Staubli VAL3: StaubliUI.pjx

--- StaubliUI.pjx ---
Parameters version=s7.3 stackSize=15000 millimeterUnit=true
Program file=Bool_Edit.pgx
Program file=BoolMess_Edit.pgx
Program file=Control_Action.pgx
Program file=Control_AxisPar.pgx
Program file=Control_BatPara.pgx
Program file=Control_BatPrt.pgx
Program file=Control_BatSpd.pgx
Program file=Control_Bottom.pgx
Program file=Control_BottomS.pgx
Program file=Control_CPreset.pgx
Program file=Control_Joint.pgx
Program file=Control_Lable.pgx
Program file=Control_Left.pgx
Program file=Control_LeftCut.pgx
Program file=Control_LeftS.pgx
Program file=Control_List.pgx
Program file=Control_List1S.pgx
Program file=Control_ListBS.pgx
Program file=Control_ListCls.pgx
Program file=Control_ListMC.pgx
Program file=Control_ListMCD.pgx
Program file=Control_ListS.pgx
Program file=Control_Loffset.pgx
Program file=Control_MCShow.pgx
Program file=Control_Mess.pgx
Program file=Control_Panel.pgx
Program file=Control_PanelB.pgx
Program file=Control_PanelD.pgx
Program file=Control_PanelMd.pgx
Program file=Control_PanelS.pgx
Program file=Control_PanelXY.pgx
Program file=Control_PanTitl.pgx
Program file=Control_Para.pgx
Program file=Control_Para1.pgx
Program file=Control_PatMove.pgx
Program file=Control_Point.pgx
Program file=Control_Preset.pgx
Program file=Control_Recipe.pgx
Program file=Control_Remote.pgx
Program file=Control_Scara.pgx
Program file=Control_Timer.pgx
Program file=Control_Traj.pgx
Program file=Control_YesNO.pgx
Program file=Float_Edit.pgx
Program file=Form_4jHome.pgx
Program file=Form_6jHome.pgx
Program file=Form_Action.pgx
Program file=Form_Bye.pgx
Program file=Form_Config.pgx
Program file=Form_LabelList.pgx
Program file=Form_Main.pgx
Program file=Form_MainS.pgx
Program file=Form_Panel.pgx
Program file=Form_Panel4P.pgx
Program file=Form_PanelBool.pgx
Program file=Form_PanelJoint.pgx
Program file=Form_PanelList.pgx
Program file=Form_PanelPoint.pgx
Program file=Form_PanelStr.pgx
Program file=Form_Patten.pgx
Program file=Form_PattenD.pgx
Program file=Form_PattenS.pgx
Program file=Form_Prod.pgx
Program file=Form_Product.pgx
Program file=Form_ScaraRobot.pgx
Program file=Form_SelSharp.pgx
Program file=Form_Simulation.pgx
Program file=Form_Welcome.pgx
Program file=Int_Edit.pgx
Program file=Int_EditS.pgx
Program file=Key_ListBase.pgx
Program file=Key_ListMC.pgx
Program file=ReadMe.pgx
Program file=Sel_Edit.pgx
Program file=start.pgx
Program file=stop.pgx
Program file=Str_Edit.pgx
Program file=Str_SplitChar.pgx
Program file=Str_SplitComma.pgx
Data file=StaubliUI.dtx

--- StaubliUI.dtx ---
mdesc mNomSpeed
num nPanelLTopX
num nPanelLTopY
num nPanelWidthX
num nPanelLengthY
string sBuff
string sData

--- Control_AxisPar.pgx ---
public program Control_AxisPar(num& x_nPos, num& x_nSpeed, num& x_nPrecent, num& x_nJogSpeed, bool x_bTraj)
  local string l_sItem[6]
  local num l_nNum
  local num l_nKey
  local num l_nData[6]
  local num l_nSelectIndex
begin
  //为lasman3.0进行配置
  //修改点位的参数


  //通过局部变量来实现内部存储


  l_nData[0]=x_nPos
  l_nData[1]=x_nSpeed
  l_nData[2]=x_nPrecent
  l_nData[3]=x_nJogSpeed

  l_sItem[0]="位置mm   :"+toString(".3",l_nData[0])
  l_sItem[1]="速度m/min:"+toString(".3",l_nData[1])
  l_sItem[2]="比例分度 :"+toString(".3",l_nData[2])
  l_sItem[3]="点动速度 :"+toString(".3",l_nData[3])
  call Control_BottomS(",,,,,,取消,确定")

  call Control_PanelXY(8,0,17,4)
  call Control_Panel("参数")
  call Control_List(l_sItem,l_nSelectIndex)


  //按键响应
  while true
    l_nKey=getKey()

    switch l_nKey
      case 261
        l_nSelectIndex=max(0,l_nSelectIndex-1)
      break

      case 266
        if x_bTraj
          l_nSelectIndex=min(1,l_nSelectIndex+1)
        else
           l_nSelectIndex=min(3,l_nSelectIndex+1)
        endIf

      break

      case 278

        x_nPos=l_nData[0]
        x_nSpeed=l_nData[1]
        x_nPrecent=l_nData[2]
        x_nJogSpeed=l_nData[3]
        cls()
        return
      break


      case 277,255
        cls()
        return
      break



      case 270

        call Float_Edit(l_nData[l_nSelectIndex],nPanelLTopX+11,l_nSelectIndex+nPanelLTopY+1)


        l_nData[l_nSelectIndex]=max(0,l_nData[l_nSelectIndex])
        l_nData[3]=min(100,max(0,l_nData[3]))
      break

    endSwitch

    if l_nKey!=-1
      l_sItem[0]="位置mm   :"+toString(".3",l_nData[0])
      l_sItem[1]="速度m/min:"+toString(".3",l_nData[1])
      l_sItem[2]="比例分度 :"+toString(".3",l_nData[2])
      l_sItem[3]="点动速度 :"+toString(".3",l_nData[3])
      call Control_List(l_sItem,l_nSelectIndex)

    endIf






  endWhile

end

--- Control_BatSpd.pgx ---
public program Control_BatSpd(num& x_nFrom, num& x_nTo, num& x_nSpeed, num& x_nAcc)
  local string l_sItem[4]
  local num l_nNum
  local num l_nKey
  local num l_nData[6]
  local num l_nSelectIndex
begin

  //为lasman3.0进行配置
  //批处理速度


  l_nData[0]=x_nFrom
  l_nData[1]=x_nTo
  l_nData[2]=100
  l_nData[3]=15
  l_sItem[0]="开始序号:"+toString("",l_nData[0])
  l_sItem[1]="结束序号:"+toString("",l_nData[1])
  l_sItem[2]="速度    :"+toString("",l_nData[2])
  l_sItem[3]="加速度  :"+toString("",l_nData[3])



  call Control_BottomS(",,,,,,取消,确定")
  call Control_PanelXY(8,0,15,4)
  call Control_Panel("批处理速度")
  call Control_List(l_sItem,l_nSelectIndex)
  while true
    l_nKey=getKey()

    switch l_nKey
      case 261
        l_nSelectIndex=max(0,l_nSelectIndex-1)
      break

      case 266
        l_nSelectIndex=min(l_nSelectIndex+1,3)
      break

      case 278
        x_nFrom=l_nData[0]
        x_nTo=l_nData[1]
        x_nSpeed=l_nData[2]
        x_nAcc=l_nData[3]
        cls()
        return
      break


      case 277,255

        cls()
        return
      break

      case 270

        call Float_Edit(l_nData[l_nSelectIndex],nPanelLTopX+7,l_nSelectIndex+nPanelLTopY+1)
      break

    endSwitch

    if l_nKey!=-1
  l_sItem[0]="开始序号:"+toString("",l_nData[0])
  l_sItem[1]="结束序号:"+toString("",l_nData[1])
  l_sItem[2]="速度    :"+toString("",l_nData[2])
  l_sItem[3]="加速度  :"+toString("",l_nData[3])
      call Control_List(l_sItem,l_nSelectIndex)

    endIf






  endWhile





end

--- Control_CPreset.pgx ---
public program Control_CPreset(num& x_nPreset[] (dimensions=2), trsf& x_trCut[], num x_nMax, num x_nIndex)
  local string l_sItem[6]
  local num l_nNum
  local num l_nKey
  local num l_nData[5]
  local num l_nIndex
  local num l_nBuff
  local bool l_bFirst
begin

  //为lasman3.0进行定制
  //修改工艺参数


  //  //把传入参数临时存储
  //  l_nIndex=x_trCut[x_nIndex].x
  //  for l_nNum=0 to 4
  //    l_nData[l_nNum]=x_nPreset[l_nIndex,l_nNum]
  //  endFor
  //
  //  //界面初始化
  //      l_sItem[0]="工艺号  :"+toString("",l_nIndex)
  //      l_sItem[1]="激光功率  :"+toString("",l_nData[0])
  //      l_sItem[2]="气体压力  :"+toString("",l_nData[1])
  //      l_sItem[3]="占空比频率:"+toString("",l_nData[2])
  //      l_sItem[4]="激光占空比:"+toString("",l_nData[3])
  //      l_sItem[5]="随动高度  :"+toString("",l_nData[4])
  //      call Control_List(l_sItem,l_nBuff)
   l_nIndex=x_trCut[x_nIndex].x
  call Control_BottomS(",,,,,,退出,应用")
  call Control_PanelXY(8,0,15,6)
  call Control_Panel(toString("",x_nIndex)+":工艺值")
  call Control_List(l_sItem,l_nBuff)
  //按键响应
  while true
    l_nKey=getKey()

    switch l_nKey
      case 261
        l_nIndex=max(1,l_nIndex-1)
        //l_nSelectIndex=max(0,l_nSelectIndex-1)
      break

      case 266
        l_nIndex=min(50,l_nIndex+1)
        // l_nSelectIndex=min(l_nSelectIndex+1,5)
      break

      case 264
        x_nIndex=max(0,x_nIndex-1)


      break



      case 268
        x_nIndex=min(x_nMax-1,x_nIndex+1)
         l_nIndex=x_trCut[x_nIndex].x
      break





      case 278
        //        for l_nNum=0 to 4
        //          x_nPreset[x_nIndex,l_nNum]=min(max(l_nData[l_nNum],0),100)
        //      x.x=l_nIndex
        x_trCut[x_nIndex].x=l_nIndex
     //   return
      l_nIndex=x_trCut[x_nIndex].x
      break


      case 277
        return
      break

      //      case 270
      //        call Float_Edit(l_nData[l_nSelectIndex],nPanelLTopX+12,l_nSelectIndex+nPanelLTopY+1)
      //        l_nData[l_nSelectIndex]=min(max(l_nData[l_nSelectIndex],0),100)
      //      break

    endSwitch

    if l_nKey!=-1 or !l_bFirst
      l_bFirst=true

      for l_nNum=0 to 4
        l_nData[l_nNum]=x_nPreset[l_nIndex,l_nNum]
      endFor
      for l_nNum=0 to 4
        l_nData[l_nNum]=x_nPreset[l_nIndex,l_nNum]
      endFor
         call Control_PanTitl(toString("",x_nIndex+1)+"点:工艺值")
      l_sItem[0]="工艺号    :"+toString("",l_nIndex)
      l_sItem[1]="激光功率  :"+toString("",l_nData[0])
      l_sItem[2]="气体压力  :"+toString("",l_nData[1])
      l_sItem[3]="占空比频率:"+toString("",l_nData[2])
      l_sItem[4]="激光占空比:"+toString("",l_nData[3])
      l_sItem[5]="随动高度  :"+toString("",l_nData[4])
      call Control_List(l_sItem,l_nBuff)

    endIf







  endWhile





end

--- Control_ListCls.pgx ---
program Control_ListCls()
  local num l_nIndex
begin

  //说明：
  //函数功能：把方框中进行清空




  //对方框的定义进行赋初值
  if nPanelLengthY<=0 and nPanelLTopX<=0 and nPanelLTopY<=0 and nPanelWidthX<=0
    call Control_PanelXY(20,0,18,11)
  endIf

  //清空列表
  setTextMode(0)
  for l_nIndex=0 to nPanelLengthY-1
    gotoxy(nPanelLTopX+1,nPanelLTopY+l_nIndex+1)
    put(left("                                               ",nPanelWidthX))
  endFor

  //参数判断  对于选择项的判断
  // x_nSelectItem=min(max(0,x_nSelectItem),nPanelLengthY-1)


end

--- Control_ListMC.pgx ---
public program Control_ListMC(bool& x_bMC[], num& x_nSelectItem, num x_nText)
  local num l_nIndex
  local bool l_bRes
  local string l_sText
  local num l_nFrist
begin
  //说明：
  //函数功能：在划定的框内，把选中项给显示出来
  //l_nFirst  在列表中第一个显示的项的序号
  //x_nSelectItem  被选中的项的序号
  //l_nCount 合法列表项的项总数，如何数组中间为空，则可能被截断

  l_nFrist=0
  x_nSelectItem=min(max(0,x_nSelectItem),size(x_bMC)-1)
  if x_nSelectItem>=nPanelLengthY
    l_nFrist=x_nSelectItem-nPanelLengthY+1
  endIf


  //把列表给画出来
  for l_nIndex=0 to min(nPanelLengthY-1,size(x_bMC)-l_nFrist)
    gotoxy(nPanelLTopX+1,nPanelLTopY+l_nIndex+1)
    //选中项变成黑色


    //MOVEL
    if !x_bMC[l_nIndex+l_nFrist]
      if l_nIndex+l_nFrist==x_nSelectItem

        setTextMode(1)
      else
        setTextMode(0)
      endIf
      put(left(toString("",l_nIndex+l_nFrist+1)+"       ",5 )+left("MOVEL             ",nPanelWidthX-5))
    else

      //MOVEC
      setTextMode(0)
      put(left("                                               ",nPanelWidthX))
      gotoxy(nPanelLTopX+1,nPanelLTopY+l_nIndex+1)
      if l_nIndex+l_nFrist!=x_nSelectItem
        put(left(toString("",l_nIndex+l_nFrist+1)+"       ",5 )+left("MOVEC Pc Pt              ",nPanelWidthX-5))
      else
        if x_nText==0
          setTextMode(1)
        else
          setTextMode(0)
        endIf
        put(left(toString("",l_nIndex+l_nFrist+1)+"       ",5 )+"MOVEC")
        gotoxy(nPanelLTopX+12,nPanelLTopY+l_nIndex+1)
        if x_nText==1

          setTextMode(1)
        else
          setTextMode(0)
        endIf
        put("Pc")
        //目标点
        gotoxy(nPanelLTopX+15,nPanelLTopY+l_nIndex+1)

        if x_nText==2
          setTextMode(1)
        else
          setTextMode(0)
        endIf
        put("Pt")
      endIf
    endIf
  endFor

  setTextMode(0)
  while l_nIndex< nPanelLengthY
    gotoxy(nPanelLTopX+1,nPanelLTopY+l_nIndex+1)
    put(left("                          ",nPanelWidthX-2))
    l_nIndex=l_nIndex+1
  endWhile

end

--- Control_Loffset.pgx ---
public program Control_Loffset(num& x_nFrom, num& x_nTo)
  local string l_sItem[2]
  local num l_nNum
  local num l_nKey
  local num l_nData[6]
  local num l_nSelectIndex
begin

  //为lasman3.0配置
  //局部偏差
l_nData[0]=x_nFrom
l_nData[1]=x_nTo

  l_sItem[0]="开始    :"+toString("",l_nData[0])
  l_sItem[1]="停止    :"+toString("",l_nData[1])
  call Control_BottomS(",,,,,,取消,确定")
  call Control_PanelXY(8,0,15,6)
  call Control_Panel("局部偏差值")
  call Control_List(l_sItem,l_nSelectIndex)
  while true
    l_nKey=getKey()

    switch l_nKey
      case 261
        l_nSelectIndex=max(0,l_nSelectIndex-1)
      break

      case 266
        l_nSelectIndex=min(l_nSelectIndex+1,1)
      break

      case 278
          x_nFrom=l_nData[0]
          x_nTo=l_nData[1]
         cls()
        return
      break


      case 277,255

        cls()
        return
      break

      case 270
        call Float_Edit(l_nData[l_nSelectIndex],nPanelLTopX+7,l_nSelectIndex+nPanelLTopY+1)
      break

    endSwitch

    if l_nKey!=-1
  l_sItem[0]="开始    :"+toString("",l_nData[0])
  l_sItem[1]="停止    :"+toString("",l_nData[1])
      call Control_List(l_sItem,l_nSelectIndex)

    endIf






  endWhile





end

--- Control_MCShow.pgx ---
public program Control_MCShow(num x_nIndex, num x_nMoveType)
  local string l_sS[3]
begin

  //lasman3.0
  //为圆弧进行配置

  if x_nMoveType>2 or x_nMoveType<1
    return
  endIf
  l_sS[0]=toString("",x_nIndex+1)+"."+"MoveC "
  l_sS[1]=toString("",1)+" "
  l_sS[2]=left(" "+toString("",2)+"       ",nPanelWidthX-len(l_sS[0])-len(l_sS[1]))
  setTextMode(0)
  gotoxy(nPanelLTopX+1,min(nPanelLengthY,x_nIndex+1))
  put(l_sS[0])
  setTextMode(sel(x_nMoveType==1,1,0))
  put(l_sS[1])
  setTextMode(sel(x_nMoveType==1,0,1))
  put(l_sS[2])


  setTextMode(0)

end

--- Control_PanelB.pgx ---
public program Control_PanelB(string x_sLeftTitle, string x_sRightTitle)
begin

  //画左右两个方框

  call Control_PanelS(x_sLeftTitle,0,0,18,11)

  call Control_PanelS(x_sRightTitle,20,0,18,11)

end

--- Control_PanelS.pgx ---
public program Control_PanelS(string x_sTitle, num x_nLTopX, num x_nLTopY, num x_nWidthX, num x_nLengthY)
  local num l_nIndex
begin
  //画有标题的框



  //设定框的位置与大小
  call Control_PanelXY(x_nLTopX,x_nLTopY,x_nWidthX,x_nLengthY)

  //文本显示状况进行设定
   call Control_Panel(x_sTitle)



end

--- Control_Para1.pgx ---
public program Control_Para1(trsf& x_trTrsf, bool& x_bRes, bool x_bCut, num x_nType)
  local string l_sItem[6]
  local num l_nNum
  local num l_nKey
  local num l_nData[6]
  local num l_nSelectIndex
begin
  //为lasman3.0进行配置
  //修改点位的参数


  //通过局部变量来实现内部存储
  l_nData[3]=x_trTrsf.x
  l_nData[4]=x_trTrsf.y
  l_nData[0]=x_trTrsf.z
  l_nData[1]=x_trTrsf.rx

  l_nData[2]=x_trTrsf.ry
  l_nData[5]=x_trTrsf.rz
  l_nNum=sel(x_bRes,1,0)

  //界面初始化
  resize(sData,1,2)
  if x_bCut

    sData[0]="直线"
    sData[1]="圆弧"
    l_sItem[0]="速度(mm/s:"+toString(".3",l_nData[0])
    l_sItem[1]="加速度(%):"+toString(".3",l_nData[1])
    l_sItem[2]="BLend(mm):"+toString(".3",l_nData[2])
    l_sItem[3]="工艺     :"+toString(".3",l_nData[3])
    l_sItem[4]="动作     :"+toString(".3",l_nData[4])
    l_sItem[5]="圆弧/直线:"+sData[l_nNum]

  else
    sData[0]="MoveJ"
    sData[1]="MoveL"
    l_sItem[0]="速度(mm/s:"+toString(".3",l_nData[0])
    l_sItem[1]="加速度(%):"+toString(".3",l_nData[1])
    l_sItem[2]="关节/直线:"+sData[l_nNum]

  endIf

  call Control_BottomS(",,,,,,取消,确定")
  if x_bCut
    if x_nType!=10
      call Control_PanelXY(8,0,18,5)
    else
      call Control_PanelXY(8,0,18,6)
    endIf
  else
    call Control_PanelXY(8,0,17,3)
  endIf
  call Control_Panel("参数")
  call Control_List(l_sItem,l_nSelectIndex)


  //按键响应
  while true
    l_nKey=getKey()

    switch l_nKey
      case 261
        l_nSelectIndex=max(0,l_nSelectIndex-1)
      break

      case 266
        if x_bCut
          if x_nType==10
            l_nSelectIndex=min(l_nSelectIndex+1,5)
          else
            l_nSelectIndex=min(l_nSelectIndex+1,4)
          endIf
        else
          l_nSelectIndex=min(l_nSelectIndex+1,2)
        endIf
      break

      case 278
        x_trTrsf.x=l_nData[3]
        x_trTrsf.y=l_nData[4]
        x_trTrsf.z=l_nData[0]
        x_trTrsf.rx=l_nData[1]

        x_trTrsf.ry=l_nData[2]
        x_trTrsf.rz=l_nData[5]
        x_bRes=(l_nNum==1)
        cls()
        return
      break


      case 277,255
        cls()
        return
      break



      case 270
        if (l_nSelectIndex==2 and !x_bCut) or (l_nSelectIndex==5 and x_bCut)
          call Sel_Edit(l_nNum,nPanelLTopX+11,l_nSelectIndex+nPanelLTopY+1,sData)

        else
          call Float_Edit(l_nData[l_nSelectIndex],nPanelLTopX+11,l_nSelectIndex+nPanelLTopY+1)
        endIf
      break

    endSwitch

    if l_nKey!=-1
      if x_bCut

        sData[0]="直线"
        sData[1]="圆弧"
        l_sItem[0]="速度(mm/s:"+toString(".3",l_nData[0])
        l_sItem[1]="加速度(%):"+toString(".3",l_nData[1])
        l_sItem[2]="BLend(mm):"+toString(".3",l_nData[2])
        l_sItem[3]="工艺     :"+toString(".3",l_nData[3])
        l_sItem[4]="动作     :"+toString(".3",l_nData[4])
        l_sItem[5]="圆弧/直线:"+sData[l_nNum]

      else
        sData[0]="MoveJ"
        sData[1]="MoveL"
        l_sItem[0]="速度(mm/s:"+toString(".3",l_nData[0])
        l_sItem[1]="加速度(%):"+toString(".3",l_nData[1])
        l_sItem[2]="关节/直线:"+sData[l_nNum]

      endIf
      call Control_List(l_sItem,l_nSelectIndex)

    endIf






  endWhile

end

--- Control_Point.pgx ---
public program Control_Point(pointRx& x_pP)
  local string l_sItem[6]
  local num l_nNum
  local num l_nKey
  local num l_nData[6]
  local num l_nSelectIndex
begin

  //修改点位的 Point

  l_nData[0]=x_pP.trsf.x
  l_nData[1]=x_pP.trsf.y
  l_nData[2]=x_pP.trsf.z
  l_nData[3]=x_pP.trsf.rx
  l_nData[4]=x_pP.trsf.ry
  l_nData[5]=x_pP.trsf.rz

  l_sItem[0]="X    :"+toString(".3",l_nData[0])
  l_sItem[1]="y    :"+toString(".3",l_nData[1])
  l_sItem[2]="Z    :"+toString(".3",l_nData[2])
  l_sItem[3]="RX   :"+toString(".3",l_nData[3])
  l_sItem[4]="RY   :"+toString(".3",l_nData[4])
  l_sItem[5]="RZ   :"+toString(".3",l_nData[5])

  call Control_BottomS(",,,,,,取消,确定")
  call Control_PanelXY(8,0,15,6)
  call Control_Panel("Point值")
  call Control_List(l_sItem,l_nSelectIndex)
  while true
    l_nKey=getKey()

    switch l_nKey
      case 261
        l_nSelectIndex=max(0,l_nSelectIndex-1)
      break

      case 266
        l_nSelectIndex=min(l_nSelectIndex+1,5)
      break

      case 278
        x_pP.trsf.x=l_nData[0]
        x_pP.trsf.y=l_nData[1]
        x_pP.trsf.z=l_nData[2]
        x_pP.trsf.rx=l_nData[3]
        x_pP.trsf.ry=l_nData[4]
        x_pP.trsf.rz=l_nData[5]
        cls()
        return
      break


      case 277,255

        cls()
        return
      break

      case 270
        call Float_Edit(l_nData[l_nSelectIndex],nPanelLTopX+7,l_nSelectIndex+nPanelLTopY+1)
      break

    endSwitch

    if l_nKey!=-1
      l_sItem[0]="X    :"+toString(".3",l_nData[0])
      l_sItem[1]="y    :"+toString(".3",l_nData[1])
      l_sItem[2]="Z    :"+toString(".3",l_nData[2])
      l_sItem[3]="RX   :"+toString(".3",l_nData[3])
      l_sItem[4]="RY   :"+toString(".3",l_nData[4])
      l_sItem[5]="RZ   :"+toString(".3",l_nData[5])
      call Control_List(l_sItem,l_nSelectIndex)

    endIf






  endWhile





end

--- Control_Remote.pgx ---
public program Control_Remote(num& x_nMode, num& x_nCycleCount)
  local string l_sItem[2]
  local num l_nNum
  local num l_nKey
  local num l_nData[2]
  local num l_nSelectIndex
  local string l_sSMess[6]
begin

  //为lasman3.0进行配置
  //主要是远程选择界面



  l_nData[0]=max(round(x_nMode),0)
  l_nData[1]=max(round(x_nCycleCount),0)

  l_sSMess[0]="按钮触发单工位"
  l_sSMess[1]="按钮触发单周期"
  l_sSMess[2]="按钮触发多周期"
  l_sSMess[3]="无需按钮触发"
  l_sSMess[4]="按钮触发排队"
  l_sSMess[5]="用户自定义触发"


  l_sItem[0]="生产模式:"+l_sSMess[l_nData[0]]
  l_sItem[1]="周期次数:"+toString("",l_nData[1])


  call Control_BottomS(",,,,,,取消,确定")
  call Control_PanelXY(8,0,25,2)
  call Control_ListCls()
  call Control_Panel("生产配置")
  call Control_List(l_sItem,l_nSelectIndex)
  while true
    l_nKey=getKey()

    switch l_nKey
      case 261
        l_nSelectIndex=max(0,l_nSelectIndex-1)
        //        l_nSelectIndex=l_nSelectIndex-1
        //        if l_nSelectIndex<=-1
        //          l_nSelectIndex=5
        //        endIf

      break

      case 266
        l_nSelectIndex=min(l_nSelectIndex+1,1)
        //       l_nSelectIndex=l_nSelectIndex+1
        //       if l_nSelectIndex>=6
        //        l_nSelectIndex=0
        //      endIf
      break

      case 278
        x_nMode=l_nData[0]
        x_nCycleCount=l_nData[1]

        return
      break


      case 277
        return
      break

      case 270
        if l_nSelectIndex==0
          call Sel_Edit(l_nData[0],nPanelLTopX+10,nPanelLTopY+1,l_sSMess)
        else
          call Float_Edit(l_nData[1],nPanelLTopX+10,nPanelLTopY+2)

        endIf



        l_nData[l_nSelectIndex]=max(round(l_nData[l_nSelectIndex]),0)
      break

    endSwitch

    if l_nKey!=-1
      l_sItem[0]="生产模式:"+l_sSMess[l_nData[0]]
      l_sItem[1]="周期次数:"+toString("",l_nData[1])
      call Control_List(l_sItem,l_nSelectIndex)

    endIf






  endWhile





end

--- Control_Scara.pgx ---
public program Control_Scara()
  local string l_sText[20]
  local num l_nIndex
begin
  //为Scara进行配置

//   l_sText[0]="       .:i.         "
//   l_sText[1]="         .:i.       "
//   l_sText[2]="       Xzi  iU    , "
//   l_sText[3]="     .6:     .i   : "
//   l_sText[4]="    .A    MM .E:,.n."
//   l_sText[5]="    6     8MvYIZX;v."
//   l_sText[6]="   7.     vi;iCCviX "
//   l_sText[7]="   7 :.   vtYn7Yci7 "
//   l_sText[8]="    .7Co622onU  6t; "
//   l_sText[9]="  SY7Az      .  .:Q."
//   l_sText[10]="  MMMMM           X "
//   l_sText[11]="  MM:..    "
//   l_sText[12]="  MMt:;  "
//   l_sText[13]="  MMt:;  "




   l_sText[0]="         .--.           "
   l_sText[1]="      :./    \ ..   .     "
   l_sText[2]="    .:/    |::::.;:..:   "
   l_sText[3]="   ../     |::::;;:.:     "
   l_sText[4]="   ./ . ...:i:;..:::     "
   l_sText[5]="  . .i;.......  :.;      "
   l_sText[6]="   |::|           |:|             "
   l_sText[7]=" |::. .|              "
   l_sText[8]=" |::.  |               "
   l_sText[9]=" | .:::|                "
   l_sText[10]=" |  .ri|             "
   l_sText[11]=" |r72r7|            "
   l_sText[12]=" |scara|            "


for l_nIndex=0 to 9
  gotoxy(18,l_nIndex+1)
  put(left(l_sText[l_nIndex],22))
endFor
















end

--- Form_4jHome.pgx ---
public program Form_4jHome(string x_sTitle, jointRs& x_jJ)
begin
  //call Form_MainS(",,,,,记录,保存,退出")
  title(x_sTitle)

  call Form_PattenS(x_sTitle,"记录,,,,,,保存,退出","记录,,,,,,保存,退出")
  call Control_PanelXY(22,0,15,10)
  call Control_Panel("Home")
  //call con
  gotoxy(nPanelLTopX+1,nPanelLTopY+1)
  put(left("j1:"+toString(".3",x_jJ.j1)+"        ",nPanelWidthX))

  gotoxy(nPanelLTopX+1,nPanelLTopY+2)
  put(left("j2:"+toString(".3",x_jJ.j2)+"        ",nPanelWidthX))

  gotoxy(nPanelLTopX+1,nPanelLTopY+3)
  put(left("j3:"+toString(".3",x_jJ.j3)+"        ",nPanelWidthX))

  gotoxy(nPanelLTopX+1,nPanelLTopY+4)
  put(left("j4:"+toString(".3",x_jJ.j4)+"        ",nPanelWidthX))



end

--- Form_Config.pgx ---
public program Form_Config(num& x_nNum[], num& x_nPointIndex)
  local string l_sBuff[2]
  local string l_sVersion
begin
  //为lasman3.0配置
  //主要是配置界面


  l_sBuff[0]="关"
  l_sBuff[1]="开"
  //轮询
  resize(sBuff,1,40)

  sBuff[0]="工具(Tool)X  :"+toString(".3",  x_nNum[0])
  sBuff[1]="工具(Tool)Y  :"+toString(".3",x_nNum[1])
  sBuff[2]="工具(Tool)Z  :"+toString(".3",x_nNum[2])
  sBuff[3]="工具(Tool)RX :"+toString(".3",x_nNum[3])
  sBuff[4]="工具(Tool)RY :"+toString(".3",x_nNum[4])
  sBuff[5]="工具(Tool)RZ :"+toString(".3",x_nNum[5])


  sBuff[6]="回零速度(m/min):"+toString(".3",x_nNum[6])
  sBuff[7]="不拆工具示教 :"+l_sBuff[x_nNum[7]]
  sBuff[8]="示教回退(启动:"+l_sBuff[x_nNum[8]]

  sBuff[9]="PWM频率高(HZ):"+toString(".3",x_nNum[9])
  sBuff[10]="PWM频率低(HZ):"+toString(".3",x_nNum[10])
  sBuff[11]="模拟量系数   :"+toString(".3",x_nNum[11])
  sBuff[12]="速度匹配(s)  :"+toString(".3",x_nNum[12])
  sBuff[13]="光斑补偿(mm) :"+toString(".3",x_nNum[13])


  sBuff[14]="开气延时(s)  :"+toString(".3",x_nNum[14])
  sBuff[15]="随动延时(s)  :"+toString(".3",x_nNum[15])
  sBuff[16]="工位延时(s)  :"+toString(".3",x_nNum[16])

  sBuff[17]="快捷速度(mm/s):"+toString("",x_nNum[17])
  sBuff[18]="快捷加速度(%):"+toString("",x_nNum[18])
  sBuff[19]="快捷Blend(mm):"+toString(".3",x_nNum[19])
  sBuff[20]="快捷工艺     :"+toString("",x_nNum[20])


  sBuff[21]="异步7轴(启动):"+l_sBuff[x_nNum[21]]
  sBuff[22]="7轴home点(mm):"+toString(".3",x_nNum[22])
  sBuff[23]="7轴分度      :"+toString(".3",x_nNum[23])
  sBuff[24]="7轴安全点速度:"+toString("",x_nNum[24])



  sBuff[25]="焊接(启动)   :"+l_sBuff[x_nNum[25]]
  sBuff[26]="焊接回退长度 :"+toString("",x_nNum[26])
  //sBuff[27]="步进(启动)   :"+l_sBuff[x_nNum[27]]
  sBuff[28]="步进距离(mm) :"+toString(".3",x_nNum[28])
  sBuff[29]="远程生产密码 :"+toString(".3",x_nNum[29])
  sBuff[30]="同工位多产品 :"+l_sBuff[x_nNum[30]]
  sBuff[27]="报警延时触发 :"+toString(".3",x_nNum[27])
  sBuff[31]="拐角速度自适 :"+l_sBuff[x_nNum[31]]


  sBuff[32]="异步8轴(启动):"+l_sBuff[x_nNum[32]]
  sBuff[33]="8轴home点(mm):"+toString(".3",x_nNum[33])
  sBuff[34]="8轴分度      :"+toString(".3",x_nNum[34])
  sBuff[35]="8轴安全点速度:"+toString("",x_nNum[35])

  sBuff[36]="工位完成IO输出:"+l_sBuff[x_nNum[36]]
  sBuff[37]="PLC控制外部轴:"+l_sBuff[x_nNum[37]]
  sBuff[38]="切割厚板模式 :"+l_sBuff[x_nNum[38]]


  call Control_LeftS(",,,,,上传,保存,退出,")
  call Control_PanelS("选项",17,0,20,10)
  call Control_BottomS(",,,,,上传,保存,退出,")
  call Control_List(sBuff,x_nPointIndex)


end

--- Form_Main.pgx ---
public program Form_Main(string& x_sBottomList[])
  local num l_nIndex
begin
  //欢迎界面，显示日期和时间
 userPage()
cls()
 call Control_PanelMd("RobotPolish软件主界面")



//     for l_nIndex=0 to min(7,size(x_sBottomList)-1)
//    gotoxy(1+l_nIndex*5,13)
//    if size(x_sBottomList)>l_nIndex and x_sBottomList[l_nIndex]!=""
//      put(x_sBottomList[l_nIndex])
//    endIf
//    endFor
 call Control_Bottom(x_sBottomList)
end

--- Form_MainS.pgx ---
public program Form_MainS(string x_sBottomList)
  local num l_nIndex
  local bool l_bRes
  local string l_sBuff[20]
begin
  //把字符串给分开，使用,作为分隔符
  //主界面
  call Str_SplitComma(l_bRes,x_sBottomList,l_sBuff)
  if !l_bRes
    return
  endIf
   call Form_Main(l_sBuff)
end

--- Form_PanelJoint.pgx ---
public program Form_PanelJoint(string x_sTitle, string x_sPanelTitle, jointRs& x_jJ[], num& x_nSelectIndex, string x_sBottom)
  local num l_nNum
begin

//×××××××××××××××××××××××××××××××××××××××××××××××××
//×××××××××××××××××××××××××××××××××××××××××××××××××
//if size(x_bList)!=size(x_sList)
//  return
//endIf
resize(sBuff,1,size(x_jJ))

for l_nNum=0 to size(sBuff)-1
//  if x_bList[l_nNum]
//    sBuff[l_nNum]=toString("",l_nNum+1)+"."+x_sList[l_nNum]
//  else
    sBuff[l_nNum]=toString("",l_nNum+1)+"."+"Joint"
//  endIf
endFor
//*********************************************************
call Form_PanelList(x_sTitle,x_sPanelTitle,sBuff,x_nSelectIndex,x_sBottom)

cls()

end

--- Form_PanelList.pgx ---
public program Form_PanelList(string x_sTitle, string x_sPanelTitle, string& x_sList[], num& x_nSelectIndex, string x_sBottom)
begin

//cls()
title(x_sTitle)
call Control_LeftS(x_sBottom)
call Control_PanelS(x_sPanelTitle,22,0,15,10)
call Control_BottomS(x_sBottom)
call Control_List(x_sList,x_nSelectIndex)



end

--- Form_PanelPoint.pgx ---
public program Form_PanelPoint(string x_sTitle, string x_sPanelTitle, num x_nItemCount, num& x_nSelectIndex, string x_sBottom)
  local num l_nNum
begin

//×××××××××××××××××××××××××××××××××××××××××××××××××
//×××××××××××××××××××××××××××××××××××××××××××××××××
x_nItemCount=max(0,x_nItemCount)
if x_nItemCount==0

  call Form_Panel(x_sTitle,x_sPanelTitle,x_nSelectIndex,x_sBottom)

  return
endIf


resize(sBuff,1,x_nItemCount)

for l_nNum=0 to size(sBuff)-1
//  if x_bList[l_nNum]
//    sBuff[l_nNum]=toString("",l_nNum+1)+"."+x_sList[l_nNum]
//  else
    sBuff[l_nNum]=toString("",l_nNum+1)+"."+"Point"
//  endIf
endFor
//*********************************************************
call Form_PanelList(x_sTitle,x_sPanelTitle,sBuff,x_nSelectIndex,x_sBottom)

 cls()

end

--- Form_Prod.pgx ---
public program Form_Prod(string& x_sBottomList[])
  local num l_nIndex
begin
  //欢迎界面，显示日期和时间
 userPage()
cls()
 call Control_PanelMd("RobotPolish软件生产界面")



//     for l_nIndex=0 to min(7,size(x_sBottomList)-1)
//    gotoxy(1+l_nIndex*5,13)
//    if size(x_sBottomList)>l_nIndex and x_sBottomList[l_nIndex]!=""
//      put(x_sBottomList[l_nIndex])
//    endIf
//    endFor
 call Control_Bottom(x_sBottomList)
end

--- Form_Product.pgx ---
public program Form_Product(string x_sTitle, string& x_sLableList[], string& x_sList[], string x_sBottom)
  local num l_nNum
begin

//cls()
title(x_sTitle)
setTextMode(0)
for l_nNum=0 to size(x_sLableList)-1
  gotoxy(0,l_nNum+1)
  if l_nNum==2
    setTextMode(2)
  endIf
  put(left(x_sLableList[l_nNum]+"            ",18))
  setTextMode(0)
  gotoxy(22,l_nNum+1)

   put(left(x_sList[l_nNum]+"            ",18))
endFor

call Control_BottomS(x_sBottom)



end

--- Form_Welcome.pgx ---
public program Form_Welcome(string x_sTitle, bool& x_bExit)
begin
  //欢迎界面，显示日期和时间
  userPage()
  cls()
  title(x_sTitle)
  call Control_PanelMd("欢迎使用史陶比尔机器人软件")

  while !x_bExit
    gotoxy(1,12)
    put(left("时间:"+getDate("%H:%M:%S"),30))
    gotoxy(1,13)
    put(left("日期:"+getDate("%Y")+"年"+getDate("%m")+"月"+getDate("%d")+"日",30))
    delay(0)
  endWhile



end

--- Key_ListMC.pgx ---
program Key_ListMC(bool& x_bRefresh, num& x_nKeyValue, num& x_nSelectItem, num& x_nText)
begin

 call Key_ListBase(x_bRefresh,x_nKeyValue,x_nSelectItem)
  if x_bRefresh
     x_nText=0
    return
  endIf

    x_bRefresh=true
    switch x_nKeyValue
    //向左
    case 264
      x_nText=min(max(0,x_nText-1),2)
    break
    //向右
    case 268
      x_nText=max(min(2,x_nText+1),0)
    break

    default
      x_bRefresh=false
    break

    endSwitch




end

--- SEL_EDIT.pgx ---
public program Sel_Edit(num& x_nData, num x_nX, num x_nY, string& x_sMess[])
  local num l_nKey
  local num l_nNum
  local num l_nBuff
begin
  //说明
  //函数功能：上下进行选择
  //x_nData 被选中的字符串数组序号
  //x_sMess  可选字符串数组
  //x_nX x_nY 被选中的起始点




  //参数判断
  x_nX=min(max(0,x_nX),39)
  x_nY=min(max(0,x_nY),nPanelLTopY+nPanelLengthY)
  x_nData=max(min(x_nData,size(x_sMess)-1),0)

  l_nNum=x_nData
  l_nKey=0
  l_nBuff=l_nNum-100


  //按键选择
  while l_nKey!=270 and l_nKey!=255

    //对按键进行判断
    l_nKey=getKey()
    switch l_nKey
      //向下
      case 261
        l_nNum=l_nNum-1
        if l_nNum<=-1
          l_nNum=size(x_sMess)-1
        endIf
      break

      //向上
      case 266
        l_nNum=l_nNum+1
        if l_nNum>=size(x_sMess)
          l_nNum=0
        endIf
      break
      //回车
      case 270
        x_nData=l_nNum
        return
      break
    endSwitch

    //重新刷新界面
    if l_nBuff!=l_nNum
      l_nBuff=l_nNum
      gotoxy(x_nX,x_nY)
      setTextMode(0)
      put(left(x_sMess[l_nNum]+"           ",nPanelWidthX-x_nX+nPanelLTopX))
    endIf


  endWhile
end

--- stop.pgx ---
program stop()
begin
  //库结束
  title("")
  cls()


end

--- Str_SplitComma.pgx ---
program Str_SplitComma(bool& x_bRes, string x_sStrIn, string& x_sOut[])
begin
  //****************************************************************
  //***************************************************************
  //函数名称：SplitChar
  //用途：  用于解析字符
  //创建日期：
  //作者：
  //联系方式：
  //备注：传入的数组个数决定了其中的分配
  //版本修改说明：
  //****************************************************************
  //*****************************************************************
  call Str_SplitChar(x_bRes,x_sStrIn,",",x_sOut)
end
